Fanuc KAREL source: compact_preamble.KL

PROGRAM KB00152
%NOLOCKGROUP
VAR
P1:REAL;RESULT:INTEGER
BEGIN
P1=1.0
RESULT=ROUND(P1)
END KB00152
